{attribute 'GeneratedUsingTerminal: ER7041-3002-0021'}
{attribute addProperty BoxType "ER7041-3002-0021"}
{attribute addProperty Id "ENC_Status_compactAT %I*ENC_Status_compact_4D066E1A16STM_StatusAT %I*STM_Status_DE0D6B3712ENC_Control_compactAT %Q*ENC_Control_compact_21E2D14D6STM_ControlAT %Q*STM_Control_BA4CE3524STM_VelocityAT %Q*STM_Velocity_A47A3F412WcStateAT %I*WcState_9091E0EB2InfoDataAT %I*InfoData_6538CF5F12"}
{attribute addProperty CRC "1045162735"}
{attribute addProperty Size "54"}
TYPE ER7041_3E4BEAEF EXTENDS EtcSlaveTerminalBase_947E5A46 :
STRUCT
	{attribute addProperty Name "ENC_Status_compact"}
	ENC_Status_compact : ENC_Status_compact_4D066E1A;
	{attribute addProperty Name "STM_Status"}
	STM_Status : STM_Status_DE0D6B37;
	{attribute addProperty Name "ENC_Control_compact"}
	ENC_Control_compact : ENC_Control_compact_21E2D14D;
	{attribute addProperty Name "STM_Control"}
	STM_Control : STM_Control_BA4CE352;
	{attribute addProperty Name "STM_Velocity"}
	STM_Velocity : STM_Velocity_A47A3F41;
	{attribute addProperty Name "WcState"}
	WcState : WcState_9091E0EB;
	{attribute addProperty Name "InfoData"}
	InfoData : InfoData_6538CF5F;
END_STRUCT
END_TYPE

(* stored: Version 1.2.0.0, ProductVersion 3.1.4024.9
   DUT ER7041_3E4BEAEF: Id {0b0dc75f-b3cb-439d-8eba-e4166080277d} *)
